// SIMATIC S7-200 project (STEP 7-Micro/WIN), CPU 226 CN REL 02.01

ORGANIZATION_BLOCK 主程序:OB1
TITLE=这是我做的通过自由口通讯进行温度控制的PLC例程。我用了三种方法实现，这是方法A，供大家一起学习学习。
// 注释：PLC需要实时读取温度数据并存入内存。PLC控制加热器和冷却器，以调节反应温度，加热器和冷却器不能同时开启。系统在首次上电时，调用初始化子程序，设置通讯端口参数，配置接收参数，并附加接收完成和发送完成中断，写入本机站地址——这些参数和中断必须正确设置，否则通讯无法正常进行。
// 运行过程中，当端口空闲时，PLC启动接收操作，将指令存入接收缓冲区。接收完成后，中断触发，解析指令站地址、指令类型、数据地址指针、数据长度和BCC码，置位指令接收完成标志。随后，系统计算BCC校验码，与接收到的BCC码比较，若校验正确且结束符正确，置位BCC校验正确标志。系统检查指令站地址是否与本机站地址匹配，以确认指令有效性。
// 若指令类型为读，PLC停止接收，准备发送缓冲区，写入反馈信息，将数据地址指针指向的温度数据转换为ASCII码，计算BCC码并发送。若指令类型为写，PLC将接收缓冲区中的数据写入数据地址指针指向的地址，准备发送缓冲区，写入反馈信息并发送。发送完成后，中断触发，复位BCC校验正确标志，清零BCC计算寄存器，重置地址指针，允许再次接收。
// 此外，加热器控制始终置位，确保加热器持续工作；冷却器控制受手动开关输入控制，例如手动打开冷却器。
// 
// 
BEGIN
Network 1
LD     SM0.1                 //第一次扫描调用初始化子程序  
CALL   initialize:SBR0
?000
Network 2
LDB=   VB134, VB199          //指令中的站地址与本机站地址相符  
AB=    VB102, 5              //指令类型为读指令  
A      M0.0                  //BCC码校验正确  
CALL   Read:SBR1             //调用读子程序  


Network 3
LDB=   VB134, VB199          //指令中的站地址与本机站地址相符  
AB=    VB102, 6              //指令类型为写指令  
A      M0.0                  //BCC码校验正确  
CALL   Write:SBR2            //调用写子程序 
Network 4
LD     M0.1                  //指令接收完成后调用BCC码校验子程序  
CALL   Verify:SBR3


Network 5
LD     SM4.5                 //当端口空闲时启动RCV  
RCV    VB100, 0
Network 6
LD     SM0.0
MOVW   AIW0, VW300
/I     +50, VW300
MOVW   AIW2, VW302
/I     +50, VW302
MOVW   AIW4, VW304
/I     +50, VW304
MOVW   AIW6, VW306
/I     +50, VW306
Network 7
LD     SM0.0
=      Q0.0
Network 8
LD     I0.0
=      Q0.1
END_ORGANIZATION_BLOCK

SUBROUTINE_BLOCK initialize:SBR0
TITLE=子程序注释
BEGIN
Network 1 // 网络标题
// 网络注释
LD     SM0.0
MOVB   9, SMB30              //0口"9600,N,8,1"  
Network 2
LD     SM0.0                 //RCV指令初始化  
MOVB   16#EC, SMB87
MOVB   103, SMB88
MOVB   71, SMB89
MOVB   100, SMB92
MOVB   35, SMB94
R      SM87.2, 1
Network 3
LD     SM0.0
ATCH   RCVcomplete:INT0, 23  //连接口0接收完成的中断 
Network 4
LD     SM0.0
ATCH   XMTcomplete:INT1, 9   //连接口0发送完成的中断  
Network 5
LD     SM0.0
ENI                          //中断允许  
Network 6
LD     SM0.0
MOVB   2, VB199              //将本机站地址装入寄存器  
Network 7
LD     SM0.0
MOVD   &VB102, VD149         //装入地址指针  
MOVB   0, VB179              //BCC码寄存器清零  
MOVD   &VB156, VD181         //装入地址指针  
MOVB   0, VB180              //BCC码寄存器清零  
END_SUBROUTINE_BLOCK

SUBROUTINE_BLOCK Read:SBR1
TITLE=子程序注释
BEGIN
Network 1 // 网络标题
// 网络注释
LD     SM0.0                 //停止端口0的接收  
R      SM87.7, 1
R      M0.0, 1
RCV    VB100, 0
Network 2
LD     SM0.0                 //将数据写入发送缓冲区  
MOVB   103, VB154
MOVB   1, VB155
HTA    *VD135, VB156, 16
MOVB   26, VB174
MOVB   21, VB153
Network 3
LD     SM0.0                 //计算BCC校验码  
FOR    VW177, +1, +16
Network 4
LD     SM0.0
XORB   *VD181, VB180
Network 5
LD     SM0.0
INCD   VD181
Network 6
NEXT
Network 7
LD     SM0.0
HTA    VB180, VB172, 2       //BCC校验码写入发送缓冲区  
Network 8
LD     SM4.5                 //发送反馈信息  
XMT    VB153, 0
END_SUBROUTINE_BLOCK

SUBROUTINE_BLOCK Write:SBR2
TITLE=子程序注释
BEGIN
Network 1 // 网络标题
// 网络注释
LD     SM0.0                 //停止端口0的接收  
R      SM87.7, 1
R      M0.0, 1
RCV    VB100, 0
Network 2
LD     SM0.0                 //装入要写如数据源的地址指针  
MOVD   &VB115, VD145
Network 3
LD     SM0.0                 //写入数据  
ATH    *VD145, *VD135, VB139
Network 4
LD     SM0.0                 //指令执行的反馈信息写入发送缓冲区  
MOVB   21, VB153
MOVB   103, VB154
MOVB   2, VB155
MOVB   26, VB174
Network 5
LD     SM4.5                 //发送指令执行的反馈信息  
XMT    VB153, 0
END_SUBROUTINE_BLOCK

SUBROUTINE_BLOCK Verify:SBR3
TITLE=子程序注释
BEGIN
Network 1 // 网络标题
// 网络注释
LD     SM0.0
R      M0.1, 1               //复位verify子程序的执行条件
Network 2
LD     SM0.0                 //计算BCC码  
FOR    VW175, +1, +29
Network 3
LD     SM0.0
XORB   *VD149, VB179
Network 4
LD     SM0.0
INCD   VD149
Network 5
NEXT
Network 6
LDB=   VB179, VB140          //当BCC码校验正确时，M0.0置1  
AB=    VB133, 71
S      M0.0, 1
Network 7
LDB=   VB133, 71             //BCC码错误时发送反馈信息  
AB<>   VB179, VB140
MOVB   21, VB153
MOVB   103, VB154
MOVB   3, VB155
MOVB   26, VB174
R      SM87.7, 1
RCV    VB100, 0
XMT    VB153, 0
Network 8
LDB<>  VB133, 71             //指令格式错误或RCV超时时发送反馈信息  
MOVB   21, VB153
MOVB   103, VB154
MOVB   4, VB155
MOVB   26, VB174
R      SM87.7, 1
RCV    VB100, 0
XMT    VB153, 0
END_SUBROUTINE_BLOCK

INTERRUPT_BLOCK RCVcomplete:INT0
TITLE=中断程序注释
BEGIN
Network 1 // 网络标题
// 网络注释 
LD     SM0.0
ATH    VB103, VB134, 2       //指令译码（ASCII码到十六进制）  
ATH    VB105, VB135, 8
ATH    VB113, VB139, 2
ATH    VB131, VB140, 2
S      M0.1, 1               //置位Verify子程序的触发条件  
MOVB   0, VB179              //BCC码寄存器清零  
MOVD   &VB102, VD149         //装入地址指针
END_INTERRUPT_BLOCK

INTERRUPT_BLOCK XMTcomplete:INT1
TITLE=中断程序注释
BEGIN
Network 1 // 网络标题
// 网络注释
LD     SM0.0
R      M0.0, 1               //复位BCC校验码正确的标志位  
S      SM87.7, 1             //允许口0进行接收  
MOVB   0, VB179              //BCC校验码寄存器清零  
MOVB   0, VB180              //BCC校验码寄存器清零  
MOVD   &VB102, VD149         //重新装入地址指针  
MOVD   &VB156, VD181
MOVB   0, VB133              //接收缓冲区中存放指令结束字符的字节清零
END_INTERRUPT_BLOCK
